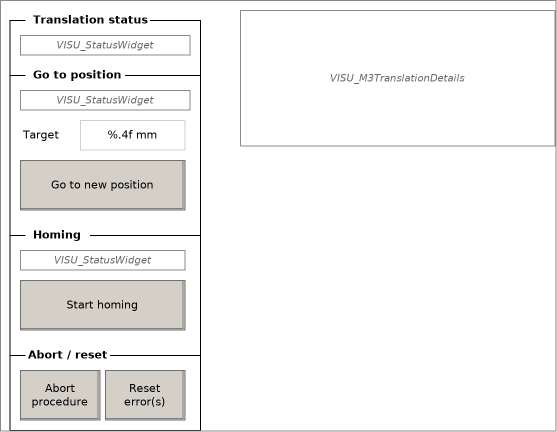
VISUALIZATION VISU_M3Translation_General  // 557x432
VAR_IN_OUT
	ref : M3Translation;
    widget : M3TranslationWidget;
END_VAR
    Button (20,160 165x50), "Go to new position", input disabled if: ref.processes.goto.statuses.enabledStatus.disabled
        OnMouseClick: execute { ref.processes.goto.do_request := TRUE; }
    Textfield (80,120 105x30), "%.4f mm", text variable: ref.processes.goto.set.position
        OnMouseClick: write the text variable via Default
    Label (20,120 55x30), "Target"
    Button (20,370 80x50), "Abort procedure", input disabled if: ref.processes.abort.statuses.enabledStatus.disabled
        OnMouseClick: execute { ref.processes.abort.do_request := TRUE; }
    Label (30,60 150x30), "Go to position"
    Line (125,75) (200,75)
    Line (10,75) (25,75)
    Line (200,20) (200,430)
    Frame (20,90 170x20)
        shows VISU_StatusWidget(widget := widget.gotoProcedureStatus)
    Button (105,370 80x50), "Reset error(s)", input disabled if: ref.processes.reset.statuses.enabledStatus.disabled
        OnMouseClick: execute { ref.processes.reset.do_request := TRUE; }
    Label (30,5 150x30), "Translation status"
    Line (150,20) (200,20)
    Line (10,20) (25,20)
    Frame (20,35 170x20)
        shows VISU_StatusWidget(widget := widget.actualStatus)
    Line (90,235) (200,235)
    Label (30,220 60x30), "Homing"
    Line (10,235) (25,235)
    Frame (20,250 165x20)
        shows VISU_StatusWidget(widget := widget.homingProcedureStatus)
    Button (20,280 165x50), "Start homing", input disabled if: ref.processes.startHoming.statuses.enabledStatus.disabled
        OnMouseClick: execute { ref.processes.startHoming.do_request := TRUE; }
    Line (10,430) (200,430)
    Line (10,430) (10,20)
    Frame (240,10 315x136)
        shows VISU_M3TranslationDetails(ref := ref)
    Line (110,355) (200,355)
    Label (25,340 85x30), "Abort / reset"
    Line (10,355) (25,355)
END_VISUALIZATION

(* stored: Version 1.1.0.1, ProductVersion 3.1.4019.2
   Visu VISU_M3Translation_General: Id {3529ca23-3af2-49f9-aa9f-f5c7eeef29f7} *)
